% RSLogix 500 project TVZ_1100_REV02.RSS, saved by version 11.00.00.00 %
PROJECT "TID_1100"    % processor: Bul.1763 MicroLogix 1100 Series A; MAIN_PROG %

PROGRAM FILES
  LAD 2 "MAIN_PROG"  7 rungs
  LAD 3 "UTILITY"  10 rungs
  LAD 4 "INSPECTION"  19 rungs
  LAD 5 "IO_COUNTER"  12 rungs
  LAD 9 "REJ TIMERS"  235 rungs
  LAD 10 "1MS_SCAN"  1 rungs
  LAD 11 "HSC0"  4 rungs
  LAD 12 "EII_COUNTS"  1 rungs  % count events to determine speed %
  LAD 13 "STI_SPEED"  6 rungs  % calc line speed based on eii counts %

DATA FILES
  O0 OUTPUT  4 elements
  I1 INPUT  6 elements
  S2 STATUS  66 elements
  B3 BINARY  5 elements
  T4 TIMER  24 elements
  C5 COUNTER  10 elements
  R6 CONTROL  1 elements
  N7 INTEGER  50 elements
  F8 FLOAT  2 elements
  B11 BITSHIFT1  255 elements
  B13 WORKBITS1  10 elements
  T14 TIMERS1  10 elements
  C15 COUNTERS1  10 elements
  R16 CTRLREGS1  10 elements
  N17 INTEGERS1  12 elements
  F18 FLOATS1  50 elements
  ST19   10 elements
  B93 TEMP BITS  100 elements  % just in case %
  T94 TEMP TMRS  100 elements  % just in case %
  C95 TEMP CTRS  100 elements  % just in case %
  R96 TEMP CTRL  100 elements  % just in case %
  N97 TEMP INTS  100 elements  % just in case %
  F98 TEMP FLTS  100 elements  % just in case %
  MG100 MSG  10 elements
  B103 TIMEDBITS  50 elements  % Bits used for 100 timed rejections %
  T104 TIMEDTMRS  115 elements  % Timers used for 100 timed rejections %

LADDER 2 "MAIN_PROG"
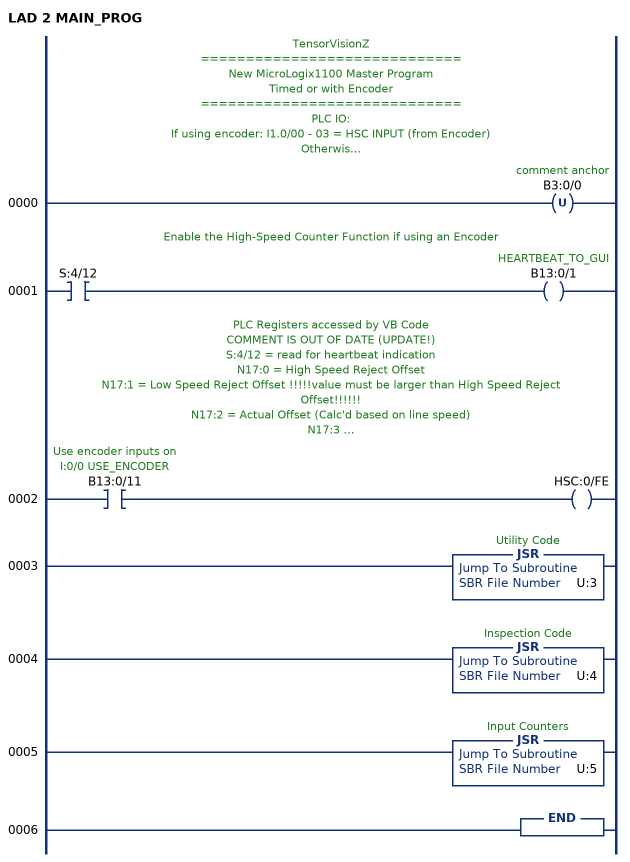
% Rung: 0 %
% TensorVisionZ
% =============================
% New MicroLogix1100 Master Program
% Timed or with Encoder
% =============================
% PLC IO:
% If using encoder: I1.0/00 - 03 = HSC INPUT (from Encoder)
% Otherwise
% I:0/0 = Encoder Pulse        O:0/0 = Rejector Output (pulse duration via timer)
% I:0/1 = Inspect Trigger       O:0/1 = Linestop Output
% I:0/2 = Reject Trigger         O:0/2 = Red Lamp
% I:0/3 = Reject Confirm        O:0/3 = Green Lamp
% I:0/4 = Pass1                     O:0/4 = Power Cycle Cameras
% I:0/5 = Fail1A                     O:0/5 = not used
% I:0/6 = Fail1B                     O:0/6 = not used
% I:0/7 = Pass2                     O:0/7 = not used
% I:0/8 = Fail2A
% i:0/9 = Fail2B %
SOR OTU B3:0/0 EOR
%   B3:0/0  "comment anchor" %
% Rung: 1 %
% Enable the High-Speed Counter Function if using an Encoder %
SOR XIC S:4/12 OTE B13:0/1 EOR
%   B13:0/1  HEARTBEAT_TO_GUI %
% Rung: 2 %
% PLC Registers accessed by VB Code
% COMMENT IS OUT OF DATE (UPDATE!)
%     S:4/12 = read for heartbeat indication
%     N17:0 = High Speed Reject Offset
%     N17:1 = Low Speed Reject Offset !!!!!value must be larger than High Speed Reject Offset!!!!!!
%     N17:2 = Actual Offset (Calc'd based on line speed)
%     N17:3 =
%     N17:4 =
%     N17:5 = Rejection Pulse Duration (in milliseconds)
%     N17:6 =
%     N17:7 = not used
%     N7:11 = Encoder Hi Preset %
SOR XIC B13:0/11 OTE HSC:0/FE EOR
%   B13:0/11  USE_ENCODER  "Use encoder inputs on I:0/0" %
% Rung: 3 %
SOR JSR U:3 EOR
%   U:3  "Utility Code" %
% Rung: 4 %
SOR JSR U:4 EOR
%   U:4  "Inspection Code" %
% Rung: 5 %
SOR JSR U:5 EOR
%   U:5  "Input Counters" %
% Rung: 6 %
SOR END EOR

LADDER 3 "UTILITY"
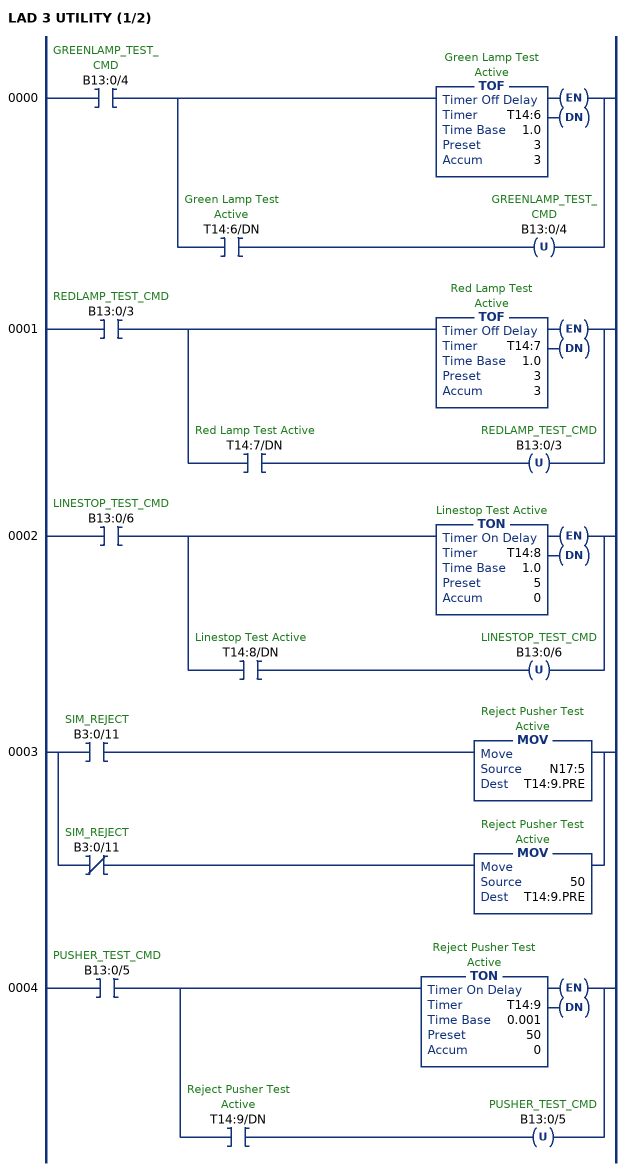
% Rung: 0 %
SOR XIC B13:0/4 BST TOF T14:6 1.0 3 3 NXB XIC T14:6/DN OTU B13:0/4 BND EOR
%   B13:0/4  GREENLAMP_TEST_CMD %
%   T14:6  "Green Lamp Test Active" %
% Rung: 1 %
SOR XIC B13:0/3 BST TOF T14:7 1.0 3 3 NXB XIC T14:7/DN OTU B13:0/3 BND EOR
%   B13:0/3  REDLAMP_TEST_CMD %
%   T14:7  "Red Lamp Test Active" %
% Rung: 2 %
SOR XIC B13:0/6 BST TON T14:8 1.0 5 0 NXB XIC T14:8/DN OTU B13:0/6 BND EOR
%   B13:0/6  LINESTOP_TEST_CMD %
%   T14:8  "Linestop Test Active" %
% Rung: 3 %
SOR BST XIC B3:0/11 MOV N17:5 T14:9.PRE NXB XIO B3:0/11 MOV 50 T14:9.PRE BND EOR
%   B3:0/11  SIM_REJECT %
%   N17:5  REJECTOR_DURATION_SP %
%   T14:9  "Reject Pusher Test Active" %
% Rung: 4 %
SOR XIC B13:0/5 BST TON T14:9 0.001 50 0 NXB XIC T14:9/DN OTU B13:0/5 BND EOR
%   B13:0/5  PUSHER_TEST_CMD %
%   T14:9  "Reject Pusher Test Active" %

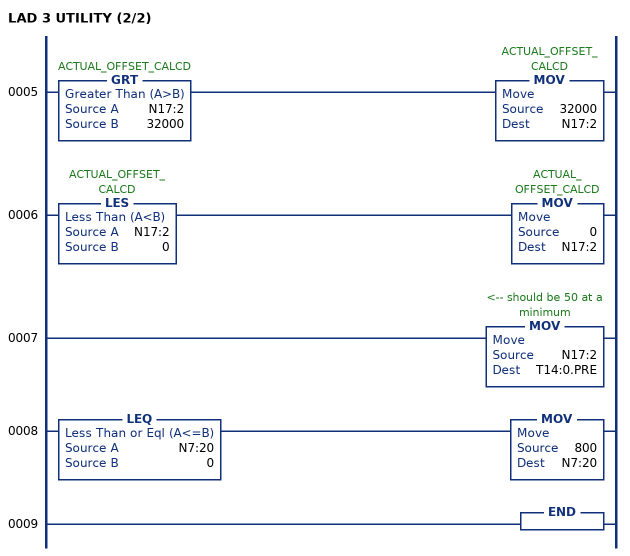
% Rung: 5 %
SOR GRT N17:2 32000 MOV 32000 N17:2 EOR
%   N17:2  ACTUAL_OFFSET_CALCD %
% Rung: 6 %
SOR LES N17:2 0 MOV 0 N17:2 EOR
%   N17:2  ACTUAL_OFFSET_CALCD %
% Rung: 7 %
SOR MOV N17:2 T14:0.PRE EOR
%   N17:2  ACTUAL_OFFSET_CALCD %
%   T14:0.PRE  "<-- should be 50 at a minimum" %
% Rung: 8 %
SOR LEQ N7:20 0 MOV 800 N7:20 EOR
% Rung: 9 %
SOR END EOR

LADDER 4 "INSPECTION"
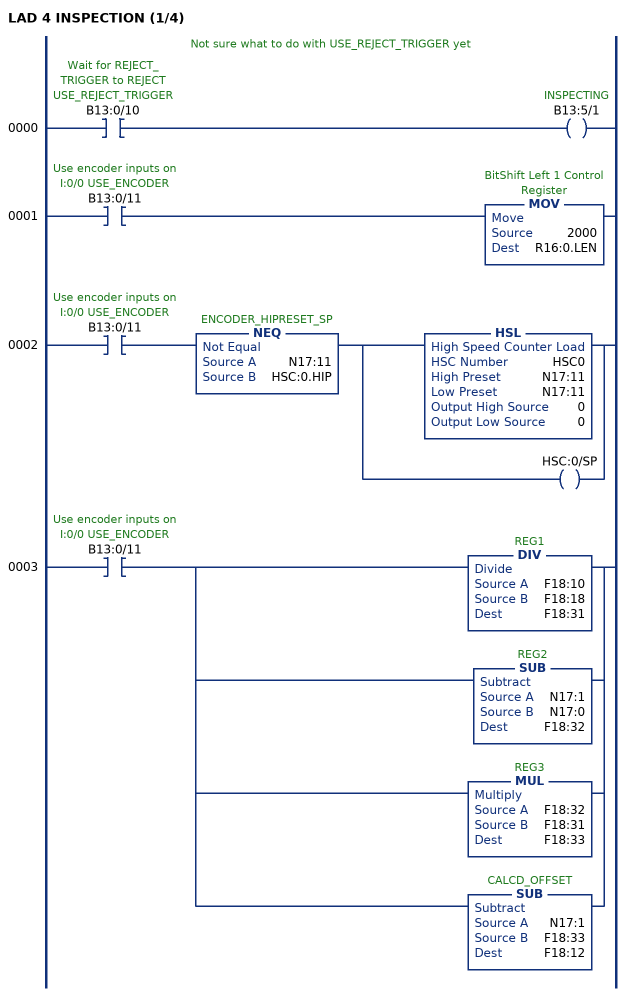
% Rung: 0 %
% Not sure what to do with USE_REJECT_TRIGGER yet %
SOR XIC B13:0/10 OTE B13:5/1 EOR
%   B13:0/10  USE_REJECT_TRIGGER  "Wait for REJECT_TRIGGER to REJECT" %
%   B13:5/1  INSPECTING %
% Rung: 1 %
SOR XIC B13:0/11 MOV 2000 R16:0.LEN EOR
%   B13:0/11  USE_ENCODER  "Use encoder inputs on I:0/0" %
%   R16:0  "BitShift Left 1 Control Register" %
% Rung: 2 %
SOR XIC B13:0/11 NEQ N17:11 HSC:0.HIP BST HSL HSC0 N17:11 N17:11 0 0 NXB OTE HSC:0/SP BND EOR
%   B13:0/11  USE_ENCODER  "Use encoder inputs on I:0/0" %
%   N17:11  ENCODER_HIPRESET_SP %
% Rung: 3 %
SOR XIC B13:0/11 BST DIV F18:10 F18:18 F18:31 NXB SUB N17:1 N17:0 F18:32 NXB MUL F18:32 F18:31 F18:33 NXB SUB N17:1 F18:33 F18:12 BND EOR
%   B13:0/11  USE_ENCODER  "Use encoder inputs on I:0/0" %
%   F18:10  AVE_LINESPEED %
%   F18:18  HISPEED_RPM_SP %
%   F18:31  REG1 %
%   N17:1  LOSPEED_OFFSET_SP %
%   N17:0  HISPEED_OFFSET_SP %
%   F18:32  REG2 %
%   F18:33  REG3 %
%   F18:12  CALCD_OFFSET %

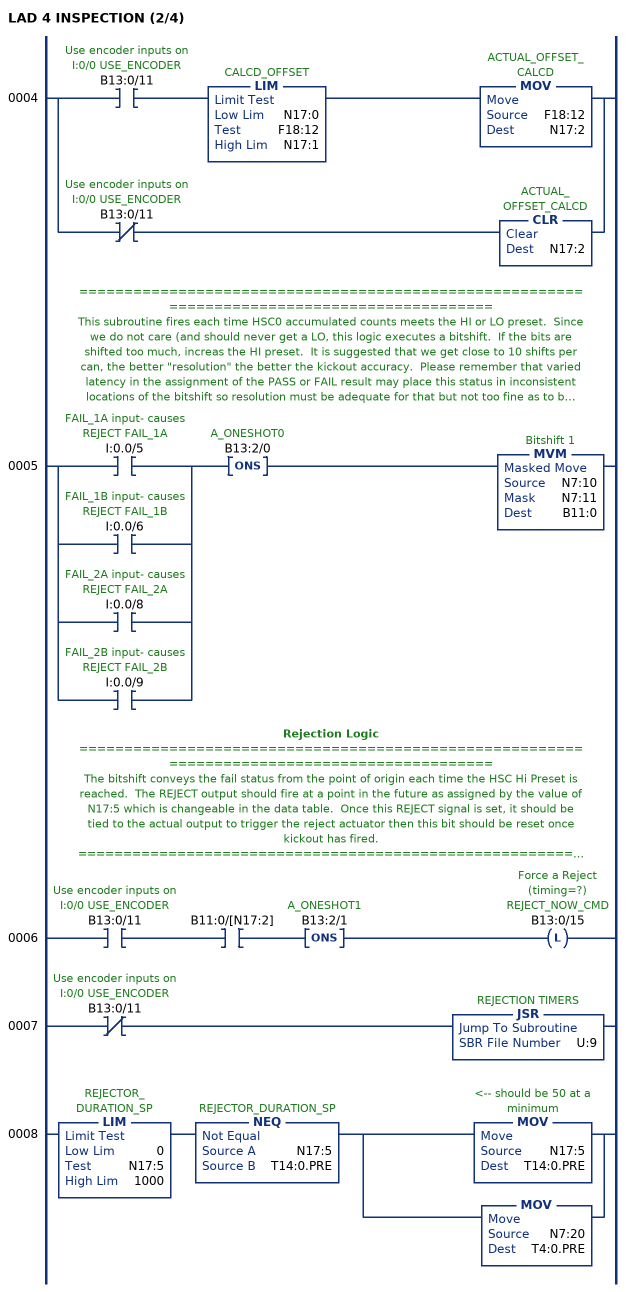
% Rung: 4 %
SOR BST XIC B13:0/11 LIM N17:0 F18:12 N17:1 MOV F18:12 N17:2 NXB XIO B13:0/11 CLR N17:2 BND EOR
%   B13:0/11  USE_ENCODER  "Use encoder inputs on I:0/0" %
%   N17:0  HISPEED_OFFSET_SP %
%   F18:12  CALCD_OFFSET %
%   N17:1  LOSPEED_OFFSET_SP %
%   N17:2  ACTUAL_OFFSET_CALCD %
% Rung: 5 %
% ============================================================================================
% This subroutine fires each time HSC0 accumulated counts meets the HI or LO preset.  Since we do not care (and should never get a LO, this logic executes a bitshift.  If the bits are shifted too much, increas the HI preset.  It is suggested that we get close to 10 shifts per can, the better "resolution" the better the kickout accuracy.  Please remember that varied latency in the assignment of the PASS or FAIL result may place this status in inconsistent locations of the bitshift so resolution must be adequate for that but not too fine as to be shift intensive.
% ============================================================================================ %
SOR BST XIC I:0.0/5 NXB XIC I:0.0/6 NXB XIC I:0.0/8 NXB XIC I:0.0/9 BND ONS B13:2/0 MVM N7:10 N7:11 B11:0 EOR
%   I:0.0/5  FAIL_1A  "FAIL_1A input- causes REJECT" %
%   I:0.0/6  FAIL_1B  "FAIL_1B input- causes REJECT" %
%   I:0.0/8  FAIL_2A  "FAIL_2A input- causes REJECT" %
%   I:0.0/9  FAIL_2B  "FAIL_2B input- causes REJECT" %
%   B13:2/0  A_ONESHOT0 %
%   N7:10  ""-1" CONSTANT" %
%   N7:11  "BSL Load Mask Bits" %
%   B11:0  "Bitshift 1" %
% Rung: 6 %
% TITLE: Rejection Logic %
% ============================================================================================
% The bitshift conveys the fail status from the point of origin each time the HSC Hi Preset is reached.  The REJECT output should fire at a point in the future as assigned by the value of N17:5 which is changeable in the data table.  Once this REJECT signal is set, it should be tied to the actual output to trigger the reject actuator then this bit should be reset once kickout has fired.
% ============================================================================================ %
SOR XIC B13:0/11 XIC B11:0/[N17:2] ONS B13:2/1 OTL B13:0/15 EOR
%   B13:0/11  USE_ENCODER  "Use encoder inputs on I:0/0" %
%   B11:0  "Bitshift 1" %
%   N17:2  ACTUAL_OFFSET_CALCD %
%   B13:2/1  A_ONESHOT1 %
%   B13:0/15  REJECT_NOW_CMD  "Force a Reject (timing=?)" %
% Rung: 7 %
SOR XIO B13:0/11 JSR U:9 EOR
%   B13:0/11  USE_ENCODER  "Use encoder inputs on I:0/0" %
%   U:9  "REJECTION TIMERS" %
% Rung: 8 %
SOR LIM 0 N17:5 1000 NEQ N17:5 T14:0.PRE BST MOV N17:5 T14:0.PRE NXB MOV N7:20 T4:0.PRE BND EOR
%   N17:5  REJECTOR_DURATION_SP %
%   T14:0.PRE  "<-- should be 50 at a minimum" %

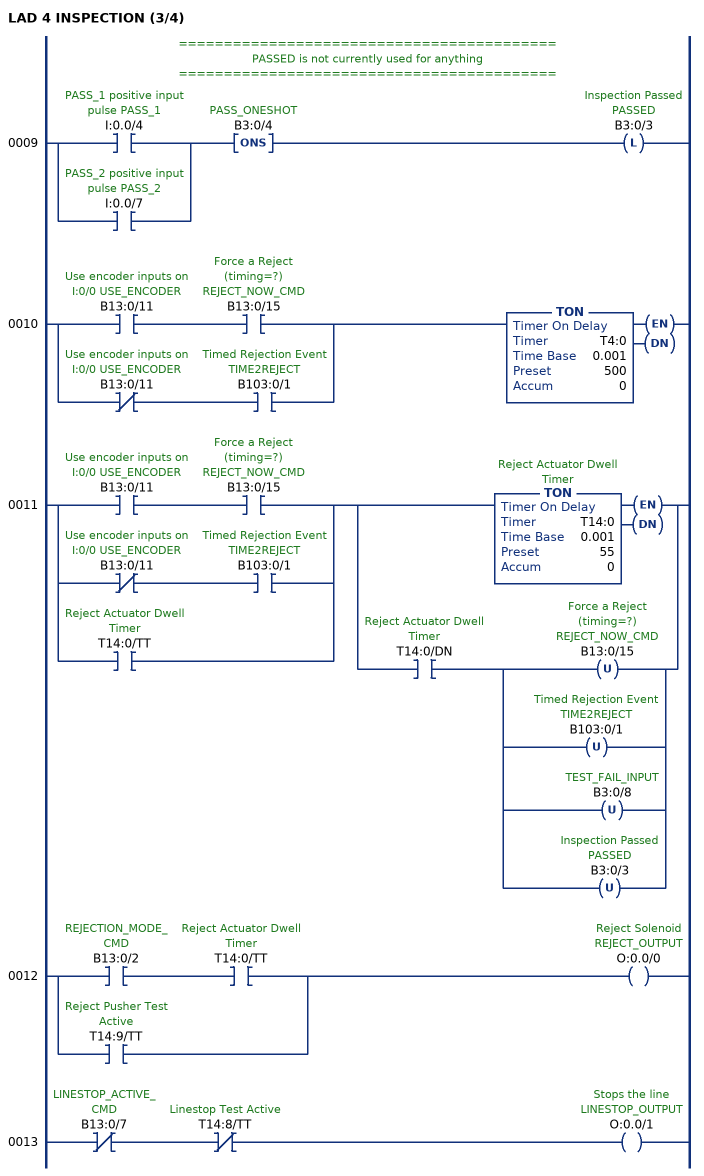
% Rung: 9 %
% ==========================================
% PASSED is not currently used for anything
% ========================================== %
SOR BST XIC I:0.0/4 NXB XIC I:0.0/7 BND ONS B3:0/4 OTL B3:0/3 EOR
%   I:0.0/4  PASS_1  "PASS_1 positive input pulse" %
%   I:0.0/7  PASS_2  "PASS_2 positive input pulse" %
%   B3:0/4  PASS_ONESHOT %
%   B3:0/3  PASSED  "Inspection Passed" %
% Rung: 10 %
SOR BST XIC B13:0/11 XIC B13:0/15 NXB XIO B13:0/11 XIC B103:0/1 BND TON T4:0 0.001 500 0 EOR
%   B13:0/11  USE_ENCODER  "Use encoder inputs on I:0/0" %
%   B13:0/15  REJECT_NOW_CMD  "Force a Reject (timing=?)" %
%   B103:0/1  TIME2REJECT  "Timed Rejection Event" %
% Rung: 11 %
SOR BST XIC B13:0/11 XIC B13:0/15 NXB XIO B13:0/11 XIC B103:0/1 NXB XIC T14:0/TT BND BST TON T14:0 0.001 55 0 NXB XIC T14:0/DN BST OTU B13:0/15 NXB OTU B103:0/1 NXB OTU B3:0/8 NXB OTU B3:0/3 BND BND EOR
%   B13:0/11  USE_ENCODER  "Use encoder inputs on I:0/0" %
%   B13:0/15  REJECT_NOW_CMD  "Force a Reject (timing=?)" %
%   B103:0/1  TIME2REJECT  "Timed Rejection Event" %
%   T14:0  "Reject Actuator Dwell Timer" %
%   B3:0/8  TEST_FAIL_INPUT %
%   B3:0/3  PASSED  "Inspection Passed" %
% Rung: 12 %
SOR BST XIC B13:0/2 XIC T14:0/TT NXB XIC T14:9/TT BND OTE O:0.0/0 EOR
%   B13:0/2  REJECTION_MODE_CMD %
%   T14:0  "Reject Actuator Dwell Timer" %
%   T14:9  "Reject Pusher Test Active" %
%   O:0.0/0  REJECT_OUTPUT  "Reject Solenoid" %
% Rung: 13 %
SOR XIO B13:0/7 XIO T14:8/TT OTE O:0.0/1 EOR
%   B13:0/7  LINESTOP_ACTIVE_CMD %
%   T14:8  "Linestop Test Active" %
%   O:0.0/1  LINESTOP_OUTPUT  "Stops the line" %

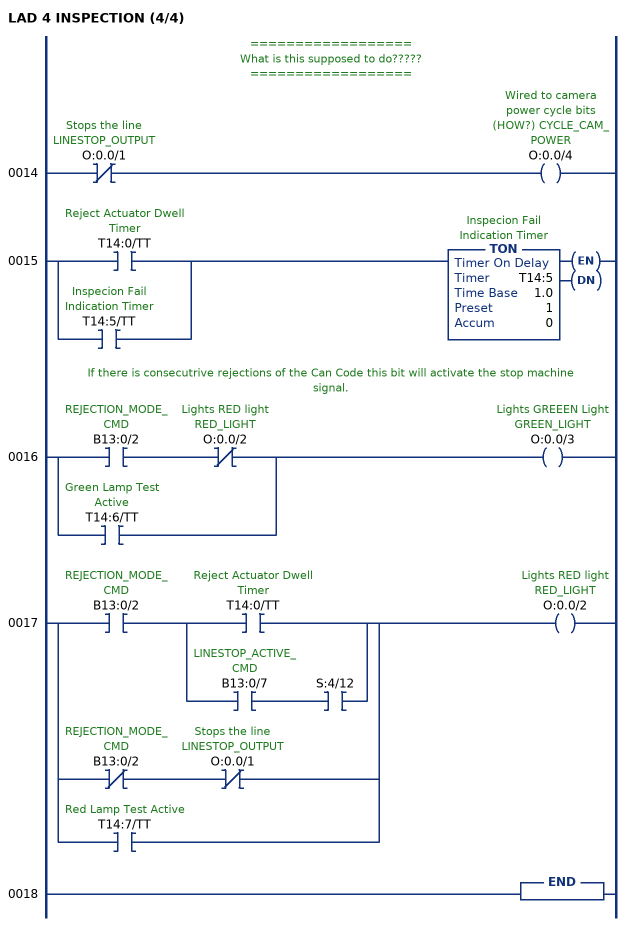
% Rung: 14 %
% ==================
% What is this supposed to do?????
% ================== %
SOR XIO O:0.0/1 OTE O:0.0/4 EOR
%   O:0.0/1  LINESTOP_OUTPUT  "Stops the line" %
%   O:0.0/4  CYCLE_CAM_POWER  "Wired to camera power cycle bits (HOW?)" %
% Rung: 15 %
SOR BST XIC T14:0/TT NXB XIC T14:5/TT BND TON T14:5 1.0 1 0 EOR
%   T14:0  "Reject Actuator Dwell Timer" %
%   T14:5  "Inspecion Fail Indication Timer" %
% Rung: 16 %
% If there is consecutrive rejections of the Can Code this bit will activate the stop machine signal. %
SOR BST XIC B13:0/2 XIO O:0.0/2 NXB XIC T14:6/TT BND OTE O:0.0/3 EOR
%   B13:0/2  REJECTION_MODE_CMD %
%   O:0.0/2  RED_LIGHT  "Lights RED light" %
%   T14:6  "Green Lamp Test Active" %
%   O:0.0/3  GREEN_LIGHT  "Lights GREEEN Light" %
% Rung: 17 %
SOR BST XIC B13:0/2 BST XIC T14:0/TT NXB XIC B13:0/7 XIC S:4/12 BND NXB XIO B13:0/2 XIO O:0.0/1 NXB XIC T14:7/TT BND OTE O:0.0/2 EOR
%   B13:0/2  REJECTION_MODE_CMD %
%   T14:0  "Reject Actuator Dwell Timer" %
%   B13:0/7  LINESTOP_ACTIVE_CMD %
%   O:0.0/1  LINESTOP_OUTPUT  "Stops the line" %
%   T14:7  "Red Lamp Test Active" %
%   O:0.0/2  RED_LIGHT  "Lights RED light" %
% Rung: 18 %
SOR END EOR

LADDER 5 "IO_COUNTER"
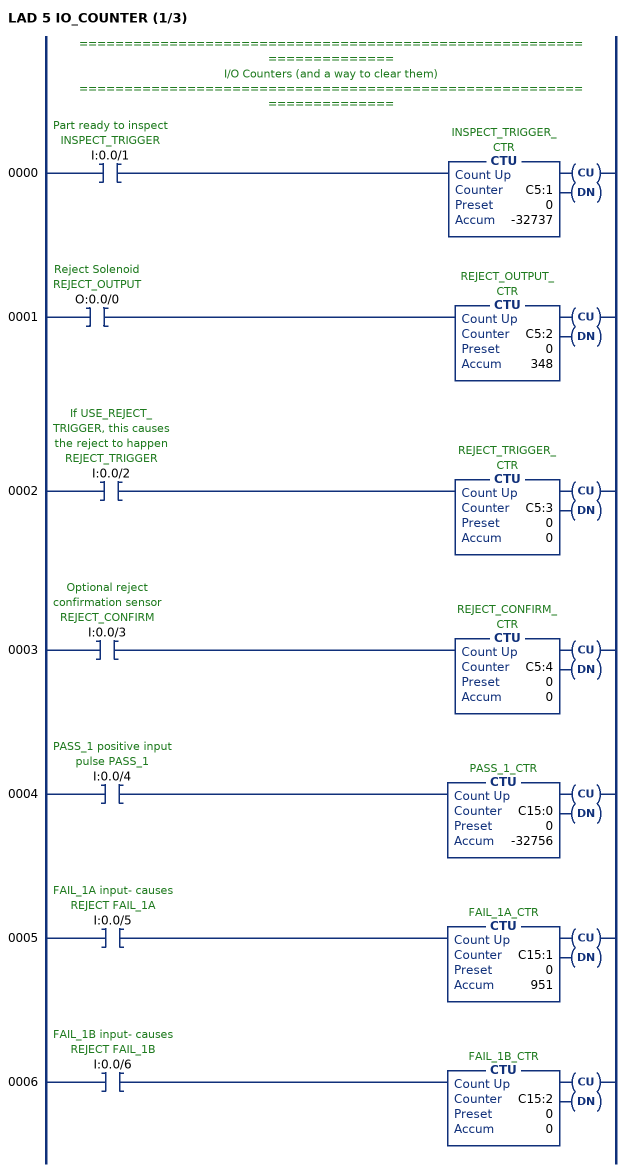
% Rung: 0 %
% ======================================================================
% I/O Counters (and a way to clear them)
% ====================================================================== %
SOR XIC I:0.0/1 CTU C5:1 0 -32737 EOR
%   I:0.0/1  INSPECT_TRIGGER  "Part ready to inspect" %
%   C5:1  INSPECT_TRIGGER_CTR %
% Rung: 1 %
SOR XIC O:0.0/0 CTU C5:2 0 348 EOR
%   O:0.0/0  REJECT_OUTPUT  "Reject Solenoid" %
%   C5:2  REJECT_OUTPUT_CTR %
% Rung: 2 %
SOR XIC I:0.0/2 CTU C5:3 0 0 EOR
%   I:0.0/2  REJECT_TRIGGER  "If USE_REJECT_TRIGGER, this causes the reject to happen" %
%   C5:3  REJECT_TRIGGER_CTR %
% Rung: 3 %
SOR XIC I:0.0/3 CTU C5:4 0 0 EOR
%   I:0.0/3  REJECT_CONFIRM  "Optional reject confirmation sensor" %
%   C5:4  REJECT_CONFIRM_CTR %
% Rung: 4 %
SOR XIC I:0.0/4 CTU C15:0 0 -32756 EOR
%   I:0.0/4  PASS_1  "PASS_1 positive input pulse" %
%   C15:0  PASS_1_CTR %
% Rung: 5 %
SOR XIC I:0.0/5 CTU C15:1 0 951 EOR
%   I:0.0/5  FAIL_1A  "FAIL_1A input- causes REJECT" %
%   C15:1  FAIL_1A_CTR %
% Rung: 6 %
SOR XIC I:0.0/6 CTU C15:2 0 0 EOR
%   I:0.0/6  FAIL_1B  "FAIL_1B input- causes REJECT" %
%   C15:2  FAIL_1B_CTR %

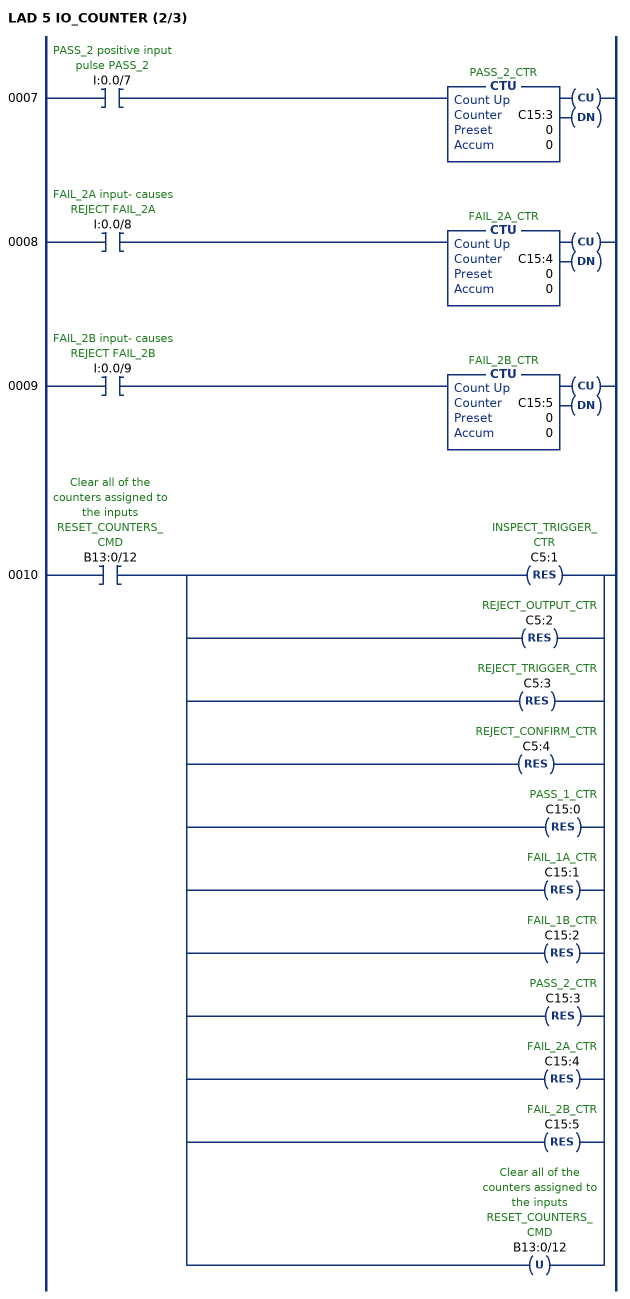
% Rung: 7 %
SOR XIC I:0.0/7 CTU C15:3 0 0 EOR
%   I:0.0/7  PASS_2  "PASS_2 positive input pulse" %
%   C15:3  PASS_2_CTR %
% Rung: 8 %
SOR XIC I:0.0/8 CTU C15:4 0 0 EOR
%   I:0.0/8  FAIL_2A  "FAIL_2A input- causes REJECT" %
%   C15:4  FAIL_2A_CTR %
% Rung: 9 %
SOR XIC I:0.0/9 CTU C15:5 0 0 EOR
%   I:0.0/9  FAIL_2B  "FAIL_2B input- causes REJECT" %
%   C15:5  FAIL_2B_CTR %
% Rung: 10 %
SOR XIC B13:0/12 BST RES C5:1 NXB RES C5:2 NXB RES C5:3 NXB RES C5:4 NXB RES C15:0 NXB RES C15:1 NXB RES C15:2 NXB RES C15:3 NXB RES C15:4 NXB RES C15:5 NXB OTU B13:0/12 BND EOR
%   B13:0/12  RESET_COUNTERS_CMD  "Clear all of the counters assigned to the inputs" %
%   C5:1  INSPECT_TRIGGER_CTR %
%   C5:2  REJECT_OUTPUT_CTR %
%   C5:3  REJECT_TRIGGER_CTR %
%   C5:4  REJECT_CONFIRM_CTR %
%   C15:0  PASS_1_CTR %
%   C15:1  FAIL_1A_CTR %
%   C15:2  FAIL_1B_CTR %
%   C15:3  PASS_2_CTR %
%   C15:4  FAIL_2A_CTR %
%   C15:5  FAIL_2B_CTR %

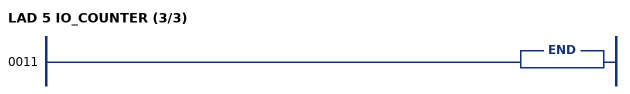
% Rung: 11 %
SOR END EOR

LADDER 9 "REJ TIMERS"
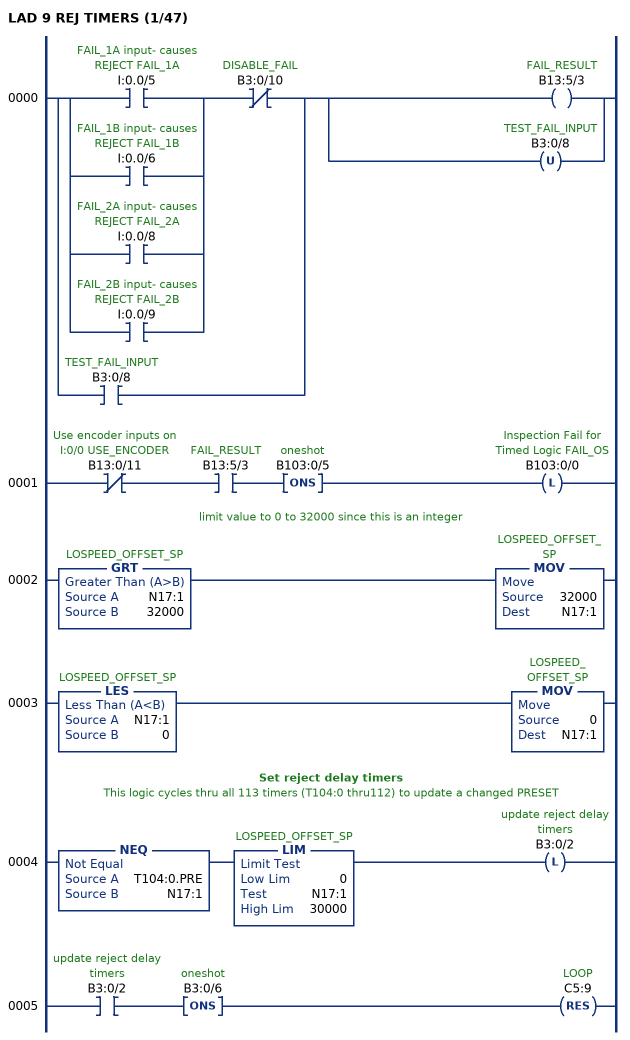
% Rung: 0 %
SOR BST BST XIC I:0.0/5 NXB XIC I:0.0/6 NXB XIC I:0.0/8 NXB XIC I:0.0/9 BND XIO B3:0/10 NXB XIC B3:0/8 BND BST OTE B13:5/3 NXB OTU B3:0/8 BND EOR
%   I:0.0/5  FAIL_1A  "FAIL_1A input- causes REJECT" %
%   I:0.0/6  FAIL_1B  "FAIL_1B input- causes REJECT" %
%   I:0.0/8  FAIL_2A  "FAIL_2A input- causes REJECT" %
%   I:0.0/9  FAIL_2B  "FAIL_2B input- causes REJECT" %
%   B3:0/10  DISABLE_FAIL %
%   B3:0/8  TEST_FAIL_INPUT %
%   B13:5/3  FAIL_RESULT %
% Rung: 1 %
SOR XIO B13:0/11 XIC B13:5/3 ONS B103:0/5 OTL B103:0/0 EOR
%   B13:0/11  USE_ENCODER  "Use encoder inputs on I:0/0" %
%   B13:5/3  FAIL_RESULT %
%   B103:0/5  "oneshot" %
%   B103:0/0  FAIL_OS  "Inspection Fail for Timed Logic" %
% Rung: 2 %
% limit value to 0 to 32000 since this is an integer %
SOR GRT N17:1 32000 MOV 32000 N17:1 EOR
%   N17:1  LOSPEED_OFFSET_SP %
% Rung: 3 %
SOR LES N17:1 0 MOV 0 N17:1 EOR
%   N17:1  LOSPEED_OFFSET_SP %
% Rung: 4 %
% TITLE: Set reject delay timers %
% This logic cycles thru all 113 timers (T104:0 thru112) to update a changed PRESET %
SOR NEQ T104:0.PRE N17:1 LIM 0 N17:1 30000 OTL B3:0/2 EOR
%   N17:1  LOSPEED_OFFSET_SP %
%   B3:0/2  "update reject delay timers" %
% Rung: 5 %
SOR XIC B3:0/2 ONS B3:0/6 RES C5:9 EOR
%   B3:0/2  "update reject delay timers" %
%   B3:0/6  "oneshot" %
%   C5:9  LOOP %

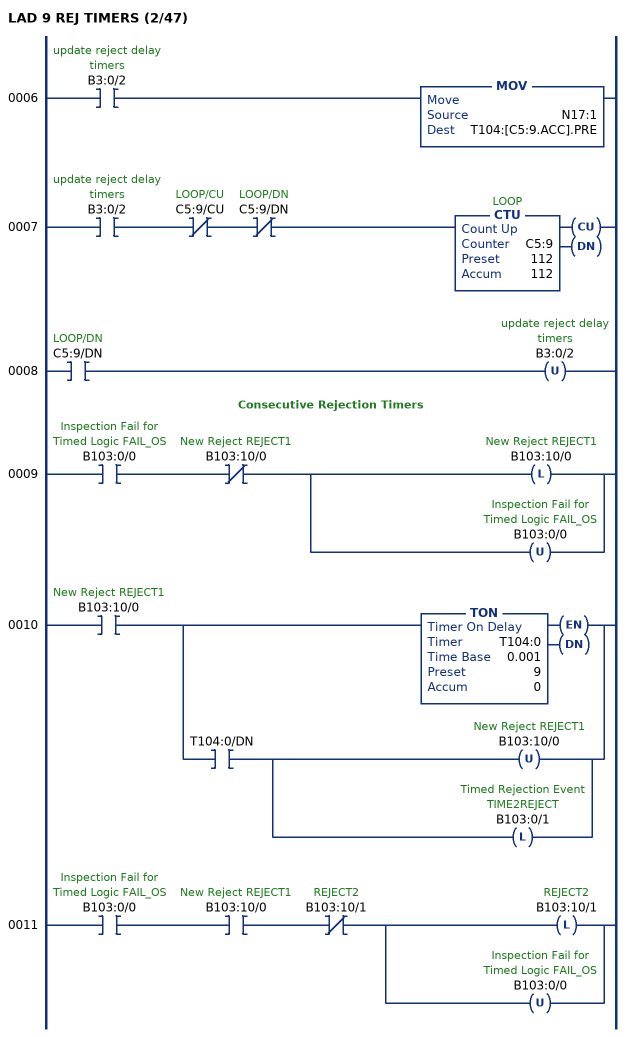
% Rung: 6 %
SOR XIC B3:0/2 MOV N17:1 T104:[C5:9.ACC].PRE EOR
%   B3:0/2  "update reject delay timers" %
%   N17:1  LOSPEED_OFFSET_SP %
%   C5:9  LOOP %
% Rung: 7 %
SOR XIC B3:0/2 XIO C5:9/CU XIO C5:9/DN CTU C5:9 112 112 EOR
%   B3:0/2  "update reject delay timers" %
%   C5:9  LOOP %
% Rung: 8 %
SOR XIC C5:9/DN OTU B3:0/2 EOR
%   C5:9  LOOP %
%   B3:0/2  "update reject delay timers" %
% Rung: 9 %
% TITLE: Consecutive Rejection Timers %
SOR XIC B103:0/0 XIO B103:10/0 BST OTL B103:10/0 NXB OTU B103:0/0 BND EOR
%   B103:0/0  FAIL_OS  "Inspection Fail for Timed Logic" %
%   B103:10/0  REJECT1  "New Reject" %
% Rung: 10 %
SOR XIC B103:10/0 BST TON T104:0 0.001 9 0 NXB XIC T104:0/DN BST OTU B103:10/0 NXB OTL B103:0/1 BND BND EOR
%   B103:10/0  REJECT1  "New Reject" %
%   B103:0/1  TIME2REJECT  "Timed Rejection Event" %
% Rung: 11 %
SOR XIC B103:0/0 XIC B103:10/0 XIO B103:10/1 BST OTL B103:10/1 NXB OTU B103:0/0 BND EOR
%   B103:0/0  FAIL_OS  "Inspection Fail for Timed Logic" %
%   B103:10/0  REJECT1  "New Reject" %
%   B103:10/1  REJECT2 %

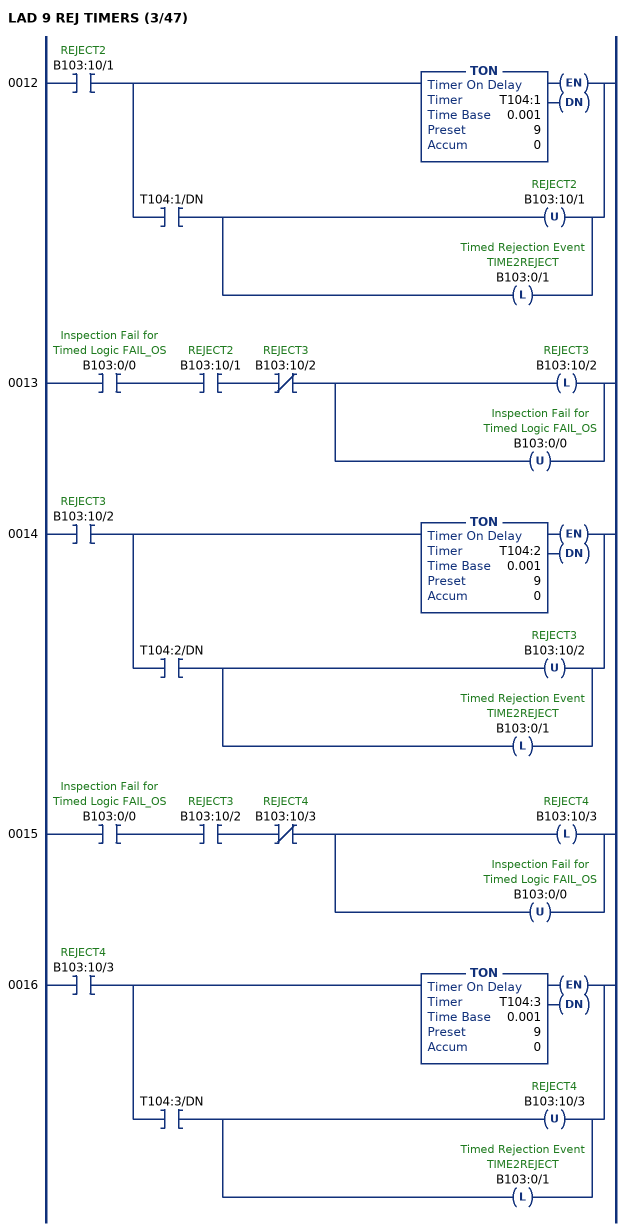
% Rung: 12 %
SOR XIC B103:10/1 BST TON T104:1 0.001 9 0 NXB XIC T104:1/DN BST OTU B103:10/1 NXB OTL B103:0/1 BND BND EOR
%   B103:10/1  REJECT2 %
%   B103:0/1  TIME2REJECT  "Timed Rejection Event" %
% Rung: 13 %
SOR XIC B103:0/0 XIC B103:10/1 XIO B103:10/2 BST OTL B103:10/2 NXB OTU B103:0/0 BND EOR
%   B103:0/0  FAIL_OS  "Inspection Fail for Timed Logic" %
%   B103:10/1  REJECT2 %
%   B103:10/2  REJECT3 %
% Rung: 14 %
SOR XIC B103:10/2 BST TON T104:2 0.001 9 0 NXB XIC T104:2/DN BST OTU B103:10/2 NXB OTL B103:0/1 BND BND EOR
%   B103:10/2  REJECT3 %
%   B103:0/1  TIME2REJECT  "Timed Rejection Event" %
% Rung: 15 %
SOR XIC B103:0/0 XIC B103:10/2 XIO B103:10/3 BST OTL B103:10/3 NXB OTU B103:0/0 BND EOR
%   B103:0/0  FAIL_OS  "Inspection Fail for Timed Logic" %
%   B103:10/2  REJECT3 %
%   B103:10/3  REJECT4 %
% Rung: 16 %
SOR XIC B103:10/3 BST TON T104:3 0.001 9 0 NXB XIC T104:3/DN BST OTU B103:10/3 NXB OTL B103:0/1 BND BND EOR
%   B103:10/3  REJECT4 %
%   B103:0/1  TIME2REJECT  "Timed Rejection Event" %

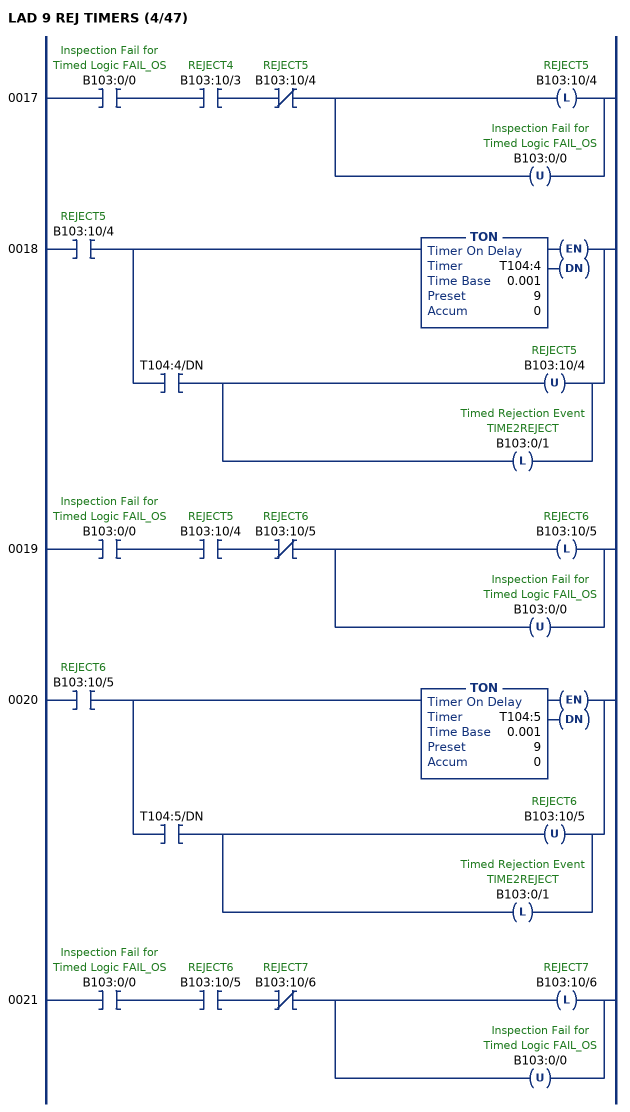
% Rung: 17 %
SOR XIC B103:0/0 XIC B103:10/3 XIO B103:10/4 BST OTL B103:10/4 NXB OTU B103:0/0 BND EOR
%   B103:0/0  FAIL_OS  "Inspection Fail for Timed Logic" %
%   B103:10/3  REJECT4 %
%   B103:10/4  REJECT5 %
% Rung: 18 %
SOR XIC B103:10/4 BST TON T104:4 0.001 9 0 NXB XIC T104:4/DN BST OTU B103:10/4 NXB OTL B103:0/1 BND BND EOR
%   B103:10/4  REJECT5 %
%   B103:0/1  TIME2REJECT  "Timed Rejection Event" %
% Rung: 19 %
SOR XIC B103:0/0 XIC B103:10/4 XIO B103:10/5 BST OTL B103:10/5 NXB OTU B103:0/0 BND EOR
%   B103:0/0  FAIL_OS  "Inspection Fail for Timed Logic" %
%   B103:10/4  REJECT5 %
%   B103:10/5  REJECT6 %
% Rung: 20 %
SOR XIC B103:10/5 BST TON T104:5 0.001 9 0 NXB XIC T104:5/DN BST OTU B103:10/5 NXB OTL B103:0/1 BND BND EOR
%   B103:10/5  REJECT6 %
%   B103:0/1  TIME2REJECT  "Timed Rejection Event" %
% Rung: 21 %
SOR XIC B103:0/0 XIC B103:10/5 XIO B103:10/6 BST OTL B103:10/6 NXB OTU B103:0/0 BND EOR
%   B103:0/0  FAIL_OS  "Inspection Fail for Timed Logic" %
%   B103:10/5  REJECT6 %
%   B103:10/6  REJECT7 %

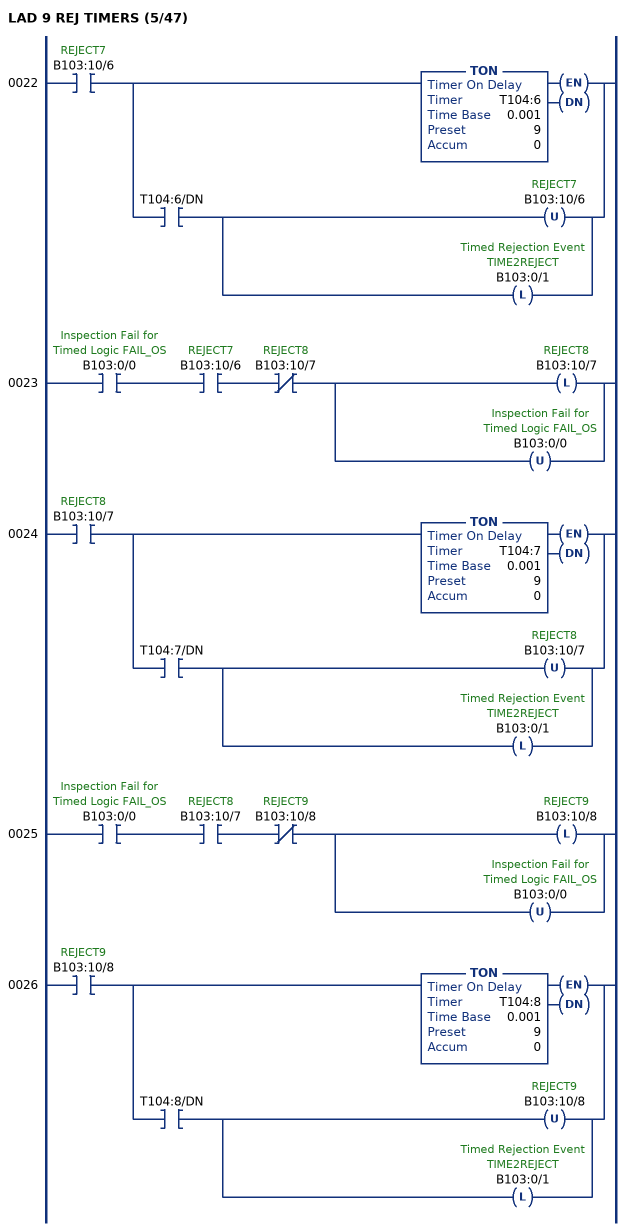
% Rung: 22 %
SOR XIC B103:10/6 BST TON T104:6 0.001 9 0 NXB XIC T104:6/DN BST OTU B103:10/6 NXB OTL B103:0/1 BND BND EOR
%   B103:10/6  REJECT7 %
%   B103:0/1  TIME2REJECT  "Timed Rejection Event" %
% Rung: 23 %
SOR XIC B103:0/0 XIC B103:10/6 XIO B103:10/7 BST OTL B103:10/7 NXB OTU B103:0/0 BND EOR
%   B103:0/0  FAIL_OS  "Inspection Fail for Timed Logic" %
%   B103:10/6  REJECT7 %
%   B103:10/7  REJECT8 %
% Rung: 24 %
SOR XIC B103:10/7 BST TON T104:7 0.001 9 0 NXB XIC T104:7/DN BST OTU B103:10/7 NXB OTL B103:0/1 BND BND EOR
%   B103:10/7  REJECT8 %
%   B103:0/1  TIME2REJECT  "Timed Rejection Event" %
% Rung: 25 %
SOR XIC B103:0/0 XIC B103:10/7 XIO B103:10/8 BST OTL B103:10/8 NXB OTU B103:0/0 BND EOR
%   B103:0/0  FAIL_OS  "Inspection Fail for Timed Logic" %
%   B103:10/7  REJECT8 %
%   B103:10/8  REJECT9 %
% Rung: 26 %
SOR XIC B103:10/8 BST TON T104:8 0.001 9 0 NXB XIC T104:8/DN BST OTU B103:10/8 NXB OTL B103:0/1 BND BND EOR
%   B103:10/8  REJECT9 %
%   B103:0/1  TIME2REJECT  "Timed Rejection Event" %

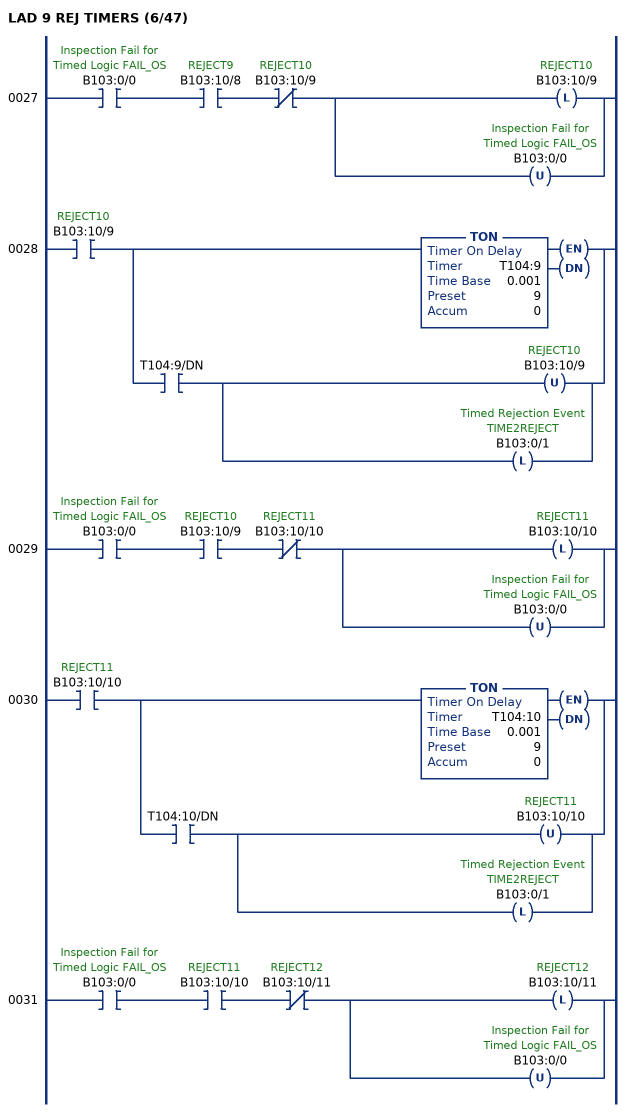
% Rung: 27 %
SOR XIC B103:0/0 XIC B103:10/8 XIO B103:10/9 BST OTL B103:10/9 NXB OTU B103:0/0 BND EOR
%   B103:0/0  FAIL_OS  "Inspection Fail for Timed Logic" %
%   B103:10/8  REJECT9 %
%   B103:10/9  REJECT10 %
% Rung: 28 %
SOR XIC B103:10/9 BST TON T104:9 0.001 9 0 NXB XIC T104:9/DN BST OTU B103:10/9 NXB OTL B103:0/1 BND BND EOR
%   B103:10/9  REJECT10 %
%   B103:0/1  TIME2REJECT  "Timed Rejection Event" %
% Rung: 29 %
SOR XIC B103:0/0 XIC B103:10/9 XIO B103:10/10 BST OTL B103:10/10 NXB OTU B103:0/0 BND EOR
%   B103:0/0  FAIL_OS  "Inspection Fail for Timed Logic" %
%   B103:10/9  REJECT10 %
%   B103:10/10  REJECT11 %
% Rung: 30 %
SOR XIC B103:10/10 BST TON T104:10 0.001 9 0 NXB XIC T104:10/DN BST OTU B103:10/10 NXB OTL B103:0/1 BND BND EOR
%   B103:10/10  REJECT11 %
%   B103:0/1  TIME2REJECT  "Timed Rejection Event" %
% Rung: 31 %
SOR XIC B103:0/0 XIC B103:10/10 XIO B103:10/11 BST OTL B103:10/11 NXB OTU B103:0/0 BND EOR
%   B103:0/0  FAIL_OS  "Inspection Fail for Timed Logic" %
%   B103:10/10  REJECT11 %
%   B103:10/11  REJECT12 %

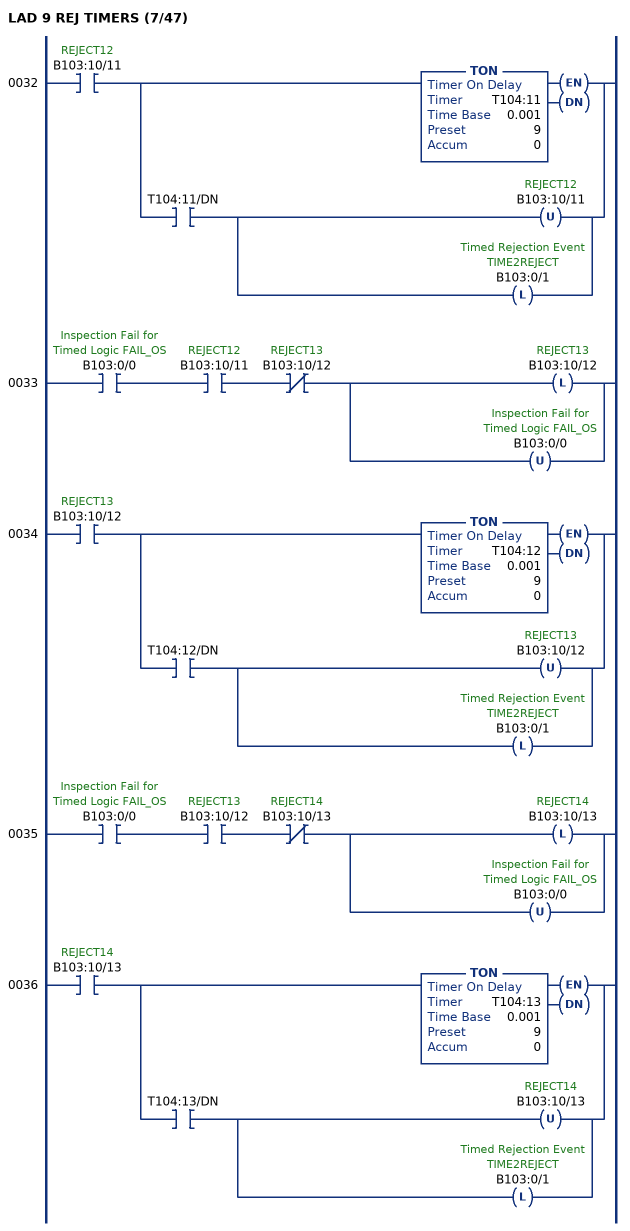
% Rung: 32 %
SOR XIC B103:10/11 BST TON T104:11 0.001 9 0 NXB XIC T104:11/DN BST OTU B103:10/11 NXB OTL B103:0/1 BND BND EOR
%   B103:10/11  REJECT12 %
%   B103:0/1  TIME2REJECT  "Timed Rejection Event" %
% Rung: 33 %
SOR XIC B103:0/0 XIC B103:10/11 XIO B103:10/12 BST OTL B103:10/12 NXB OTU B103:0/0 BND EOR
%   B103:0/0  FAIL_OS  "Inspection Fail for Timed Logic" %
%   B103:10/11  REJECT12 %
%   B103:10/12  REJECT13 %
% Rung: 34 %
SOR XIC B103:10/12 BST TON T104:12 0.001 9 0 NXB XIC T104:12/DN BST OTU B103:10/12 NXB OTL B103:0/1 BND BND EOR
%   B103:10/12  REJECT13 %
%   B103:0/1  TIME2REJECT  "Timed Rejection Event" %
% Rung: 35 %
SOR XIC B103:0/0 XIC B103:10/12 XIO B103:10/13 BST OTL B103:10/13 NXB OTU B103:0/0 BND EOR
%   B103:0/0  FAIL_OS  "Inspection Fail for Timed Logic" %
%   B103:10/12  REJECT13 %
%   B103:10/13  REJECT14 %
% Rung: 36 %
SOR XIC B103:10/13 BST TON T104:13 0.001 9 0 NXB XIC T104:13/DN BST OTU B103:10/13 NXB OTL B103:0/1 BND BND EOR
%   B103:10/13  REJECT14 %
%   B103:0/1  TIME2REJECT  "Timed Rejection Event" %

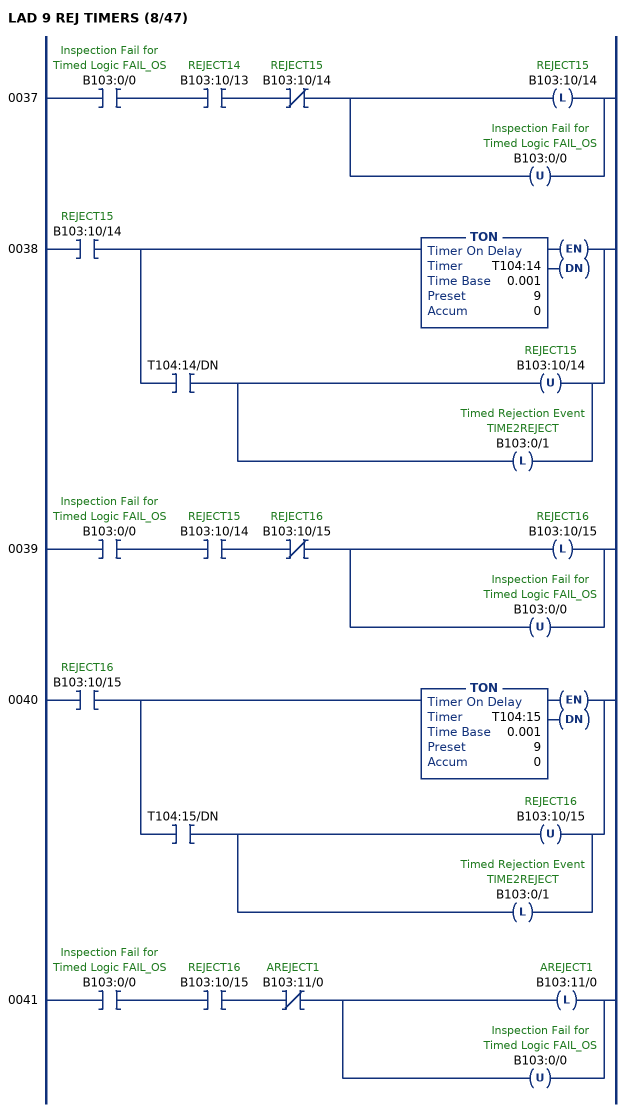
% Rung: 37 %
SOR XIC B103:0/0 XIC B103:10/13 XIO B103:10/14 BST OTL B103:10/14 NXB OTU B103:0/0 BND EOR
%   B103:0/0  FAIL_OS  "Inspection Fail for Timed Logic" %
%   B103:10/13  REJECT14 %
%   B103:10/14  REJECT15 %
% Rung: 38 %
SOR XIC B103:10/14 BST TON T104:14 0.001 9 0 NXB XIC T104:14/DN BST OTU B103:10/14 NXB OTL B103:0/1 BND BND EOR
%   B103:10/14  REJECT15 %
%   B103:0/1  TIME2REJECT  "Timed Rejection Event" %
% Rung: 39 %
SOR XIC B103:0/0 XIC B103:10/14 XIO B103:10/15 BST OTL B103:10/15 NXB OTU B103:0/0 BND EOR
%   B103:0/0  FAIL_OS  "Inspection Fail for Timed Logic" %
%   B103:10/14  REJECT15 %
%   B103:10/15  REJECT16 %
% Rung: 40 %
SOR XIC B103:10/15 BST TON T104:15 0.001 9 0 NXB XIC T104:15/DN BST OTU B103:10/15 NXB OTL B103:0/1 BND BND EOR
%   B103:10/15  REJECT16 %
%   B103:0/1  TIME2REJECT  "Timed Rejection Event" %
% Rung: 41 %
SOR XIC B103:0/0 XIC B103:10/15 XIO B103:11/0 BST OTL B103:11/0 NXB OTU B103:0/0 BND EOR
%   B103:0/0  FAIL_OS  "Inspection Fail for Timed Logic" %
%   B103:10/15  REJECT16 %
%   B103:11/0  AREJECT1 %

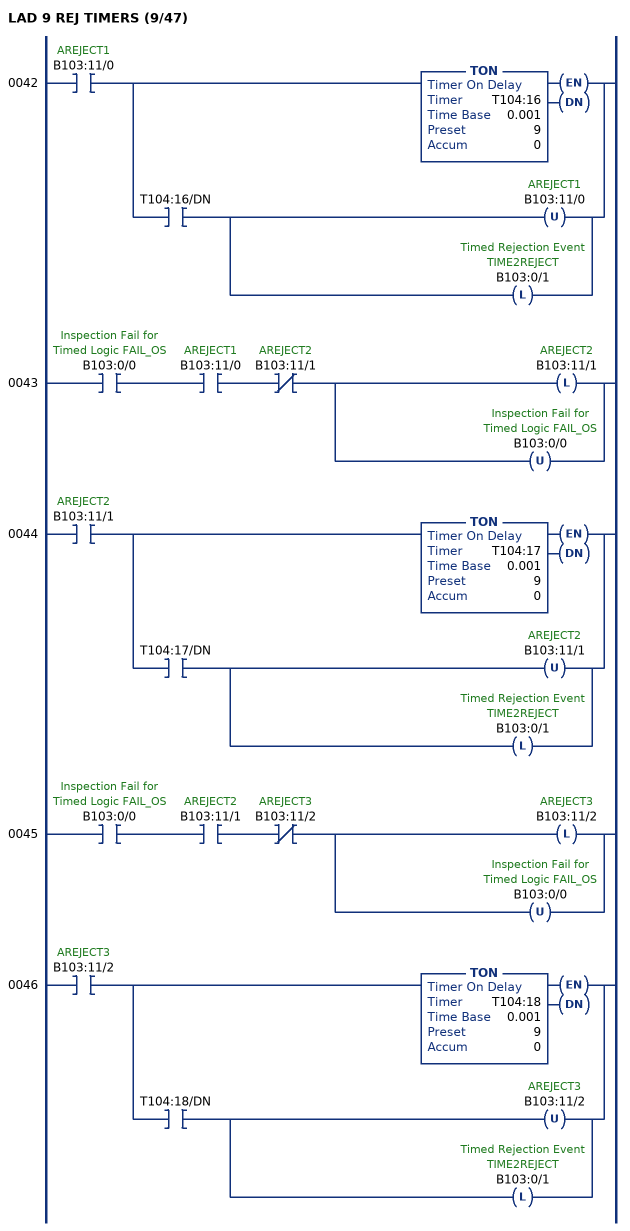
% Rung: 42 %
SOR XIC B103:11/0 BST TON T104:16 0.001 9 0 NXB XIC T104:16/DN BST OTU B103:11/0 NXB OTL B103:0/1 BND BND EOR
%   B103:11/0  AREJECT1 %
%   B103:0/1  TIME2REJECT  "Timed Rejection Event" %
% Rung: 43 %
SOR XIC B103:0/0 XIC B103:11/0 XIO B103:11/1 BST OTL B103:11/1 NXB OTU B103:0/0 BND EOR
%   B103:0/0  FAIL_OS  "Inspection Fail for Timed Logic" %
%   B103:11/0  AREJECT1 %
%   B103:11/1  AREJECT2 %
% Rung: 44 %
SOR XIC B103:11/1 BST TON T104:17 0.001 9 0 NXB XIC T104:17/DN BST OTU B103:11/1 NXB OTL B103:0/1 BND BND EOR
%   B103:11/1  AREJECT2 %
%   B103:0/1  TIME2REJECT  "Timed Rejection Event" %
% Rung: 45 %
SOR XIC B103:0/0 XIC B103:11/1 XIO B103:11/2 BST OTL B103:11/2 NXB OTU B103:0/0 BND EOR
%   B103:0/0  FAIL_OS  "Inspection Fail for Timed Logic" %
%   B103:11/1  AREJECT2 %
%   B103:11/2  AREJECT3 %
% Rung: 46 %
SOR XIC B103:11/2 BST TON T104:18 0.001 9 0 NXB XIC T104:18/DN BST OTU B103:11/2 NXB OTL B103:0/1 BND BND EOR
%   B103:11/2  AREJECT3 %
%   B103:0/1  TIME2REJECT  "Timed Rejection Event" %

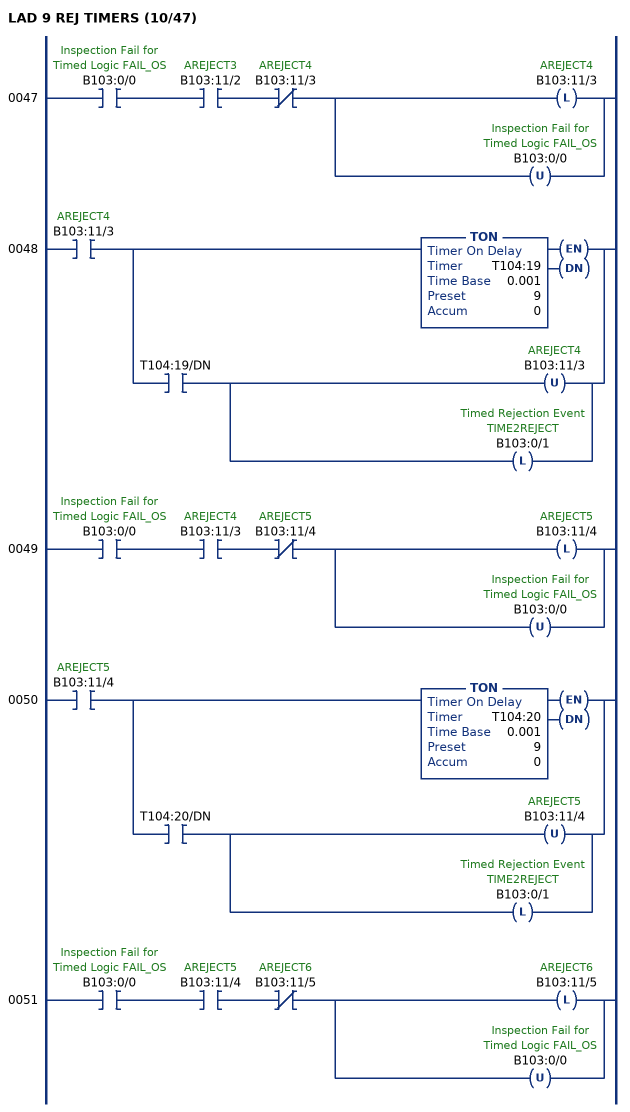
% Rung: 47 %
SOR XIC B103:0/0 XIC B103:11/2 XIO B103:11/3 BST OTL B103:11/3 NXB OTU B103:0/0 BND EOR
%   B103:0/0  FAIL_OS  "Inspection Fail for Timed Logic" %
%   B103:11/2  AREJECT3 %
%   B103:11/3  AREJECT4 %
% Rung: 48 %
SOR XIC B103:11/3 BST TON T104:19 0.001 9 0 NXB XIC T104:19/DN BST OTU B103:11/3 NXB OTL B103:0/1 BND BND EOR
%   B103:11/3  AREJECT4 %
%   B103:0/1  TIME2REJECT  "Timed Rejection Event" %
% Rung: 49 %
SOR XIC B103:0/0 XIC B103:11/3 XIO B103:11/4 BST OTL B103:11/4 NXB OTU B103:0/0 BND EOR
%   B103:0/0  FAIL_OS  "Inspection Fail for Timed Logic" %
%   B103:11/3  AREJECT4 %
%   B103:11/4  AREJECT5 %
% Rung: 50 %
SOR XIC B103:11/4 BST TON T104:20 0.001 9 0 NXB XIC T104:20/DN BST OTU B103:11/4 NXB OTL B103:0/1 BND BND EOR
%   B103:11/4  AREJECT5 %
%   B103:0/1  TIME2REJECT  "Timed Rejection Event" %
% Rung: 51 %
SOR XIC B103:0/0 XIC B103:11/4 XIO B103:11/5 BST OTL B103:11/5 NXB OTU B103:0/0 BND EOR
%   B103:0/0  FAIL_OS  "Inspection Fail for Timed Logic" %
%   B103:11/4  AREJECT5 %
%   B103:11/5  AREJECT6 %

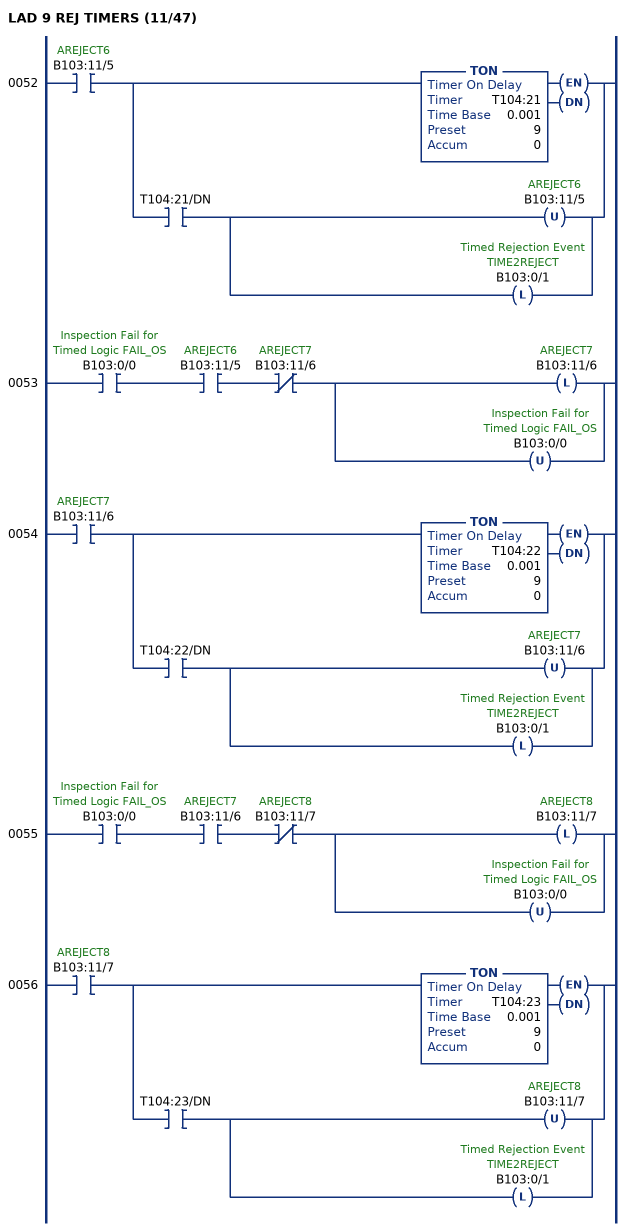
% Rung: 52 %
SOR XIC B103:11/5 BST TON T104:21 0.001 9 0 NXB XIC T104:21/DN BST OTU B103:11/5 NXB OTL B103:0/1 BND BND EOR
%   B103:11/5  AREJECT6 %
%   B103:0/1  TIME2REJECT  "Timed Rejection Event" %
% Rung: 53 %
SOR XIC B103:0/0 XIC B103:11/5 XIO B103:11/6 BST OTL B103:11/6 NXB OTU B103:0/0 BND EOR
%   B103:0/0  FAIL_OS  "Inspection Fail for Timed Logic" %
%   B103:11/5  AREJECT6 %
%   B103:11/6  AREJECT7 %
% Rung: 54 %
SOR XIC B103:11/6 BST TON T104:22 0.001 9 0 NXB XIC T104:22/DN BST OTU B103:11/6 NXB OTL B103:0/1 BND BND EOR
%   B103:11/6  AREJECT7 %
%   B103:0/1  TIME2REJECT  "Timed Rejection Event" %
% Rung: 55 %
SOR XIC B103:0/0 XIC B103:11/6 XIO B103:11/7 BST OTL B103:11/7 NXB OTU B103:0/0 BND EOR
%   B103:0/0  FAIL_OS  "Inspection Fail for Timed Logic" %
%   B103:11/6  AREJECT7 %
%   B103:11/7  AREJECT8 %
% Rung: 56 %
SOR XIC B103:11/7 BST TON T104:23 0.001 9 0 NXB XIC T104:23/DN BST OTU B103:11/7 NXB OTL B103:0/1 BND BND EOR
%   B103:11/7  AREJECT8 %
%   B103:0/1  TIME2REJECT  "Timed Rejection Event" %

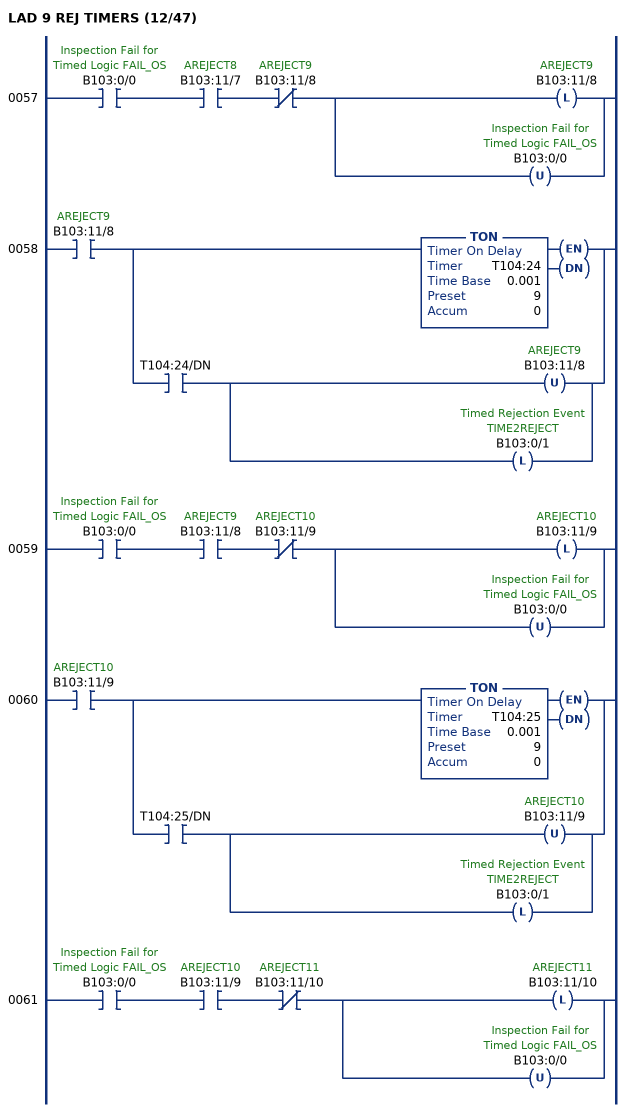
% Rung: 57 %
SOR XIC B103:0/0 XIC B103:11/7 XIO B103:11/8 BST OTL B103:11/8 NXB OTU B103:0/0 BND EOR
%   B103:0/0  FAIL_OS  "Inspection Fail for Timed Logic" %
%   B103:11/7  AREJECT8 %
%   B103:11/8  AREJECT9 %
% Rung: 58 %
SOR XIC B103:11/8 BST TON T104:24 0.001 9 0 NXB XIC T104:24/DN BST OTU B103:11/8 NXB OTL B103:0/1 BND BND EOR
%   B103:11/8  AREJECT9 %
%   B103:0/1  TIME2REJECT  "Timed Rejection Event" %
% Rung: 59 %
SOR XIC B103:0/0 XIC B103:11/8 XIO B103:11/9 BST OTL B103:11/9 NXB OTU B103:0/0 BND EOR
%   B103:0/0  FAIL_OS  "Inspection Fail for Timed Logic" %
%   B103:11/8  AREJECT9 %
%   B103:11/9  AREJECT10 %
% Rung: 60 %
SOR XIC B103:11/9 BST TON T104:25 0.001 9 0 NXB XIC T104:25/DN BST OTU B103:11/9 NXB OTL B103:0/1 BND BND EOR
%   B103:11/9  AREJECT10 %
%   B103:0/1  TIME2REJECT  "Timed Rejection Event" %
% Rung: 61 %
SOR XIC B103:0/0 XIC B103:11/9 XIO B103:11/10 BST OTL B103:11/10 NXB OTU B103:0/0 BND EOR
%   B103:0/0  FAIL_OS  "Inspection Fail for Timed Logic" %
%   B103:11/9  AREJECT10 %
%   B103:11/10  AREJECT11 %

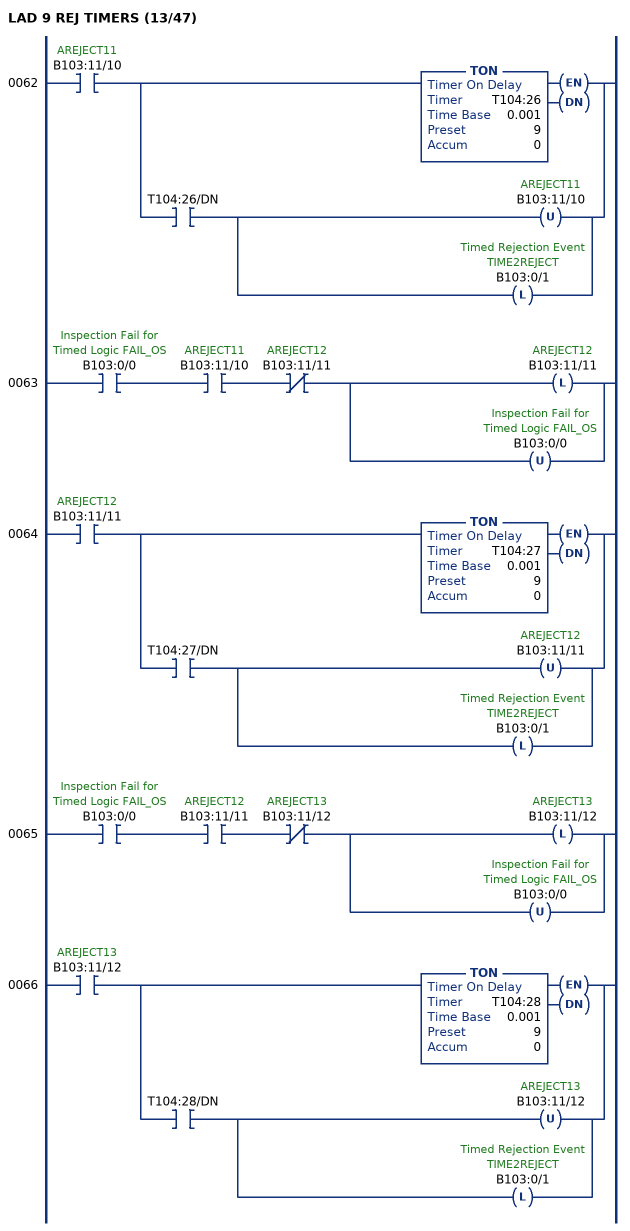
% Rung: 62 %
SOR XIC B103:11/10 BST TON T104:26 0.001 9 0 NXB XIC T104:26/DN BST OTU B103:11/10 NXB OTL B103:0/1 BND BND EOR
%   B103:11/10  AREJECT11 %
%   B103:0/1  TIME2REJECT  "Timed Rejection Event" %
% Rung: 63 %
SOR XIC B103:0/0 XIC B103:11/10 XIO B103:11/11 BST OTL B103:11/11 NXB OTU B103:0/0 BND EOR
%   B103:0/0  FAIL_OS  "Inspection Fail for Timed Logic" %
%   B103:11/10  AREJECT11 %
%   B103:11/11  AREJECT12 %
% Rung: 64 %
SOR XIC B103:11/11 BST TON T104:27 0.001 9 0 NXB XIC T104:27/DN BST OTU B103:11/11 NXB OTL B103:0/1 BND BND EOR
%   B103:11/11  AREJECT12 %
%   B103:0/1  TIME2REJECT  "Timed Rejection Event" %
% Rung: 65 %
SOR XIC B103:0/0 XIC B103:11/11 XIO B103:11/12 BST OTL B103:11/12 NXB OTU B103:0/0 BND EOR
%   B103:0/0  FAIL_OS  "Inspection Fail for Timed Logic" %
%   B103:11/11  AREJECT12 %
%   B103:11/12  AREJECT13 %
% Rung: 66 %
SOR XIC B103:11/12 BST TON T104:28 0.001 9 0 NXB XIC T104:28/DN BST OTU B103:11/12 NXB OTL B103:0/1 BND BND EOR
%   B103:11/12  AREJECT13 %
%   B103:0/1  TIME2REJECT  "Timed Rejection Event" %

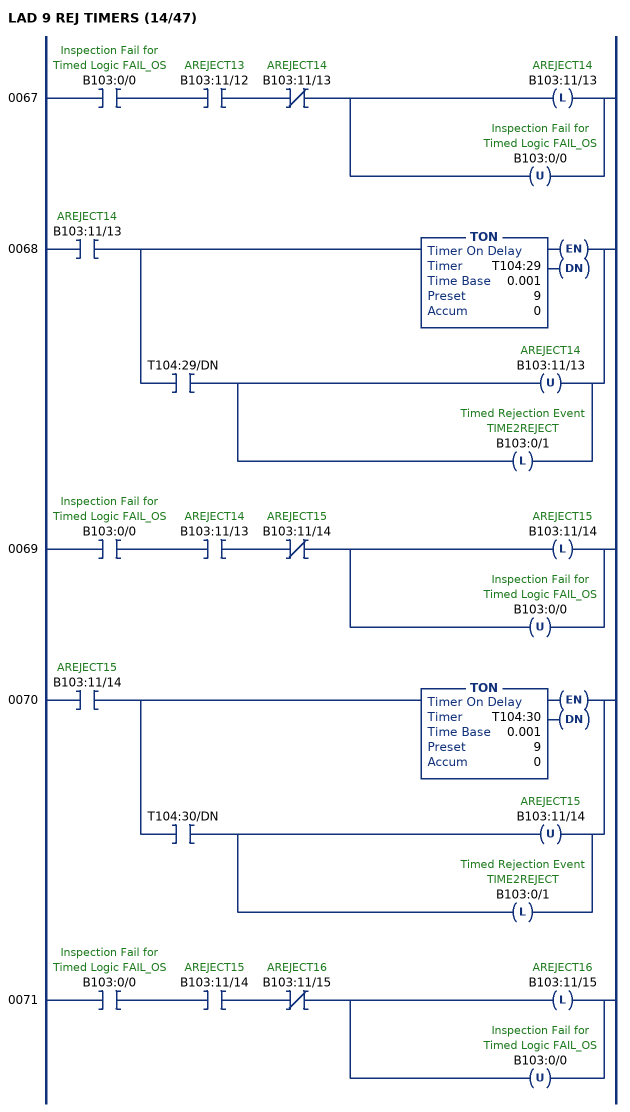
% Rung: 67 %
SOR XIC B103:0/0 XIC B103:11/12 XIO B103:11/13 BST OTL B103:11/13 NXB OTU B103:0/0 BND EOR
%   B103:0/0  FAIL_OS  "Inspection Fail for Timed Logic" %
%   B103:11/12  AREJECT13 %
%   B103:11/13  AREJECT14 %
% Rung: 68 %
SOR XIC B103:11/13 BST TON T104:29 0.001 9 0 NXB XIC T104:29/DN BST OTU B103:11/13 NXB OTL B103:0/1 BND BND EOR
%   B103:11/13  AREJECT14 %
%   B103:0/1  TIME2REJECT  "Timed Rejection Event" %
% Rung: 69 %
SOR XIC B103:0/0 XIC B103:11/13 XIO B103:11/14 BST OTL B103:11/14 NXB OTU B103:0/0 BND EOR
%   B103:0/0  FAIL_OS  "Inspection Fail for Timed Logic" %
%   B103:11/13  AREJECT14 %
%   B103:11/14  AREJECT15 %
% Rung: 70 %
SOR XIC B103:11/14 BST TON T104:30 0.001 9 0 NXB XIC T104:30/DN BST OTU B103:11/14 NXB OTL B103:0/1 BND BND EOR
%   B103:11/14  AREJECT15 %
%   B103:0/1  TIME2REJECT  "Timed Rejection Event" %
% Rung: 71 %
SOR XIC B103:0/0 XIC B103:11/14 XIO B103:11/15 BST OTL B103:11/15 NXB OTU B103:0/0 BND EOR
%   B103:0/0  FAIL_OS  "Inspection Fail for Timed Logic" %
%   B103:11/14  AREJECT15 %
%   B103:11/15  AREJECT16 %

